FUNCTION_BLOCK FB_PUMP IMPLEMENTS I_PUMP
VAR //General
	{attribute 'instance-path'} 
  {attribute 'noinit'} 
	strInstancePath:									                      STRING;
	bInit: 												                          BOOL:=TRUE;
	strFullObjectPath: 								                      STRING;
	stEvent:											                          ST_EVENT;
	bAck:												                            BOOL;	
END_VAR
VAR   // From FB_init	
	itfLogEvents: 										                      I_HANDLE_EVENTS;
  itfOpMode:											                        I_OP_MODE; 
  itfOn:                                                  I_BINARY_OUTPUT;
END_VAR                                      				
VAR	// Step chain control                				
  eSeq, eLastSeq, eNextSeq:					                      E_SEQ_ENGINE; 
                  				
  //eActiveSeqState, eLastActiveSeqState:                 E_SEQ_GENERAL;
	(*
  iInternalSeqStateCase, iLastInternalSeqStateCase:       INT:=0;       
	tonDelay, tonTimeOut, tonStepTime:						          TON;
	tDelay:													                        TIME := T#100MS;
	tTimeOut:												                        TIME := T#100MS;
	tTimeOutExt:											                      TIME := T#100MS;
	bDelayActive, bTimeOutActiveQuit, bTimeOutActiveNoQuit:	BOOL;//Timer Option
	bActiveStep, bDebugAcitve, bDebugNext:					        BOOL;//Debug Option
	i:														                          INT;
 	iError:													                        INT; //ERROR-CODE                    	                   		
	listLastSteps:											                    ARRAY[0..49] OF ST_LAST_STEPS;	
	strExtraInfo:											                      STRING; 
	eStep_Type:												                      E_STEP_STATE_TYPE; 
	bDebugModeActive:										                    BOOL;   
	bWaitForBreakpoint:										                  BOOL;
	bBreakpointActive:										                  BOOL;
	bDebugResume:											                      BOOL;   
	listBreakpoint:											                    ARRAY[0..10] OF  INT;    
*)
i:														                            INT;
stSeqCtrlGeneral:											                    ST_SEQ_CTRL_GEN;     	
END_VAR                                             		
VAR                                                 		
	bMethodeFromExtStarted:									                BOOL;
	bMethodeFromExtActive:									                BOOL;
	bMethodeFromExtDone:									                  BOOL;
	strTemp:												                        STRING;
END_VAR   
VAR
  rLimit:                                                 REAL;
END_VAR                  	
VAR_TEMP                    	
	iTemp:										                              INT;
END_VAR

// Set FBs and Interfaces ready after switch internal step
IF stSeqCtrlGeneral.iInternalSeqStateCase <> stSeqCtrlGeneral.iLastInternalSeqStateCase AND NOT stSeqCtrlGeneral.bExitSetReadyState THEN
  IF TRUE
  //AND ...
  THEN
    stSeqCtrlGeneral.bExitSetReadyState := TRUE;
  ELSE
    RETURN;
  END_IF
END_IF

stSeqCtrlGeneral.strObject := F_CreateObjectName(strInstancePath);

// First method call
_m_SequenceManager();
//_m_SaveLastStep();

CASE eSeq OF 
  E_SEQ_VALVE.BASE:;
  
	E_SEQ_ENGINE.INIT: _m_Seq_INIT();
		IF TRUE
		AND (stSeqCtrlGeneral.eActiveSeqState = E_SEQ_GENERAL.DONE) 
		THEN
			eSeq := E_SEQ_ENGINE.BASE;
		END_IF
		
	E_SEQ_ENGINE.SETUP:;
  
	// Process
  E_SEQ_ENGINE.ON: _m_Seq_ON();
    IF TRUE
		AND (stSeqCtrlGeneral.eActiveSeqState = E_SEQ_GENERAL.DONE) 
		THEN
			eSeq := E_SEQ_VALVE.BASE;
		END_IF
    
  E_SEQ_ENGINE.OFF: _m_Seq_OFF();
    IF TRUE
		AND (stSeqCtrlGeneral.eActiveSeqState = E_SEQ_GENERAL.DONE) 
		THEN
			eSeq := E_SEQ_VALVE.BASE;
		END_IF

  // End
	E_SEQ_ENGINE.END:;
	E_SEQ_ENGINE.ERROR_SEQ:;	
END_CASE

strTemp:=TO_STRING(eSeq);

METHOD PRIVATE _m_DebugManager
VAR_INPUT
	iStepID: int;
END_VAR
IF TRUE
AND THIS^.stSeqCtrlGeneral.bDebugModeActive 
AND NOT THIS^.stSeqCtrlGeneral.bActiveStep
THEN


THIS^.stSeqCtrlGeneral.bBreakpointActive:=FALSE;

FOR i:=0 TO 10 DO
	
	IF TRUE
	AND iStepID=THIS^.stSeqCtrlGeneral.listBreakpoint[i] 
	AND iStepID<>0
	THEN
		EXIT;
	END_IF
END_FOR
IF (i<=10) THEN
	THIS^.stSeqCtrlGeneral.bBreakpointActive:=TRUE;
END_IF

END_IF
END_METHOD

METHOD PRIVATE _m_Delay : BOOL
VAR_INPUT
	DelayTime:	TIME;
END_VAR
THIS^.stSeqCtrlGeneral.bDelayActive:=TRUE;
THIS^.stSeqCtrlGeneral.tDelay:=DelayTime;
_m_Delay:=FALSE;
IF THIS^.stSeqCtrlGeneral.tonDelay.Q THEN
	_m_Delay:=TRUE;
END_IF
END_METHOD

METHOD PRIVATE _m_GeneralStepSetting : BOOL
VAR_INPUT
	StepType:			    	E_STEP_STATE_TYPE;
	InfoTextID:					STRING(20);
	EnableDebug:	   			BOOL;	
	
END_VAR
IF THIS^.stSeqCtrlGeneral.bActiveStep THEN
	THIS^.stSeqCtrlGeneral.eStep_Type:=StepType;
	THIS^.stSeqCtrlGeneral.strExtraInfo:= GenLib.F_RET_TXTLIST_ENTRY(strPortNr:='851',strID:='',strTxtLstName:=InfoTextID);
END_IF
END_METHOD

METHOD PRIVATE _m_SaveLastStep : BOOL
VAR_INPUT
END_VAR
VAR
	i: dint;
END_VAR
IF NOT THIS^.stSeqCtrlGeneral.bActiveStep THEN
	
	FOR i:=49 TO 1 BY -1 DO
			stSeqCtrlGeneral.listLastSteps[i].strStepName:=stSeqCtrlGeneral.listLastSteps[i-1].strStepName;
			stSeqCtrlGeneral.listLastSteps[i].tStepTime:=stSeqCtrlGeneral.listLastSteps[i-1].tStepTime;
			stSeqCtrlGeneral.listLastSteps[i].tDelayTime:=stSeqCtrlGeneral.listLastSteps[i-1].tDelayTime;
	END_FOR
	stSeqCtrlGeneral.listLastSteps[0].strStepName:=TO_STRING(THIS^.eSeq);
	stSeqCtrlGeneral.listLastSteps[1].tStepTime:=THIS^.stSeqCtrlGeneral.tonStepTime.ET;
	stSeqCtrlGeneral.listLastSteps[1].tStepTime:=THIS^.stSeqCtrlGeneral.tonDelay.ET;
ELSE
	stSeqCtrlGeneral.listLastSteps[0].tStepTime:=THIS^.stSeqCtrlGeneral.tonStepTime.ET;
	stSeqCtrlGeneral.listLastSteps[0].tDelayTime:=THIS^.stSeqCtrlGeneral.tonDelay.ET;	
END_IF
END_METHOD

METHOD PRIVATE _m_Seq_INIT : BOOL
VAR
  ActiveSeq: STRING;
END_VAR
//THIS^._m_GeneralStepSetting(StepType:=E_STEP_STATE_TYPE.INIT,
ActiveSeq := TO_STRING(THIS^.eSeq);

CASE THIS^.stSeqCtrlGeneral.eActiveSeqState OF
E_SEQ_GENERAL.READY:;

	
E_SEQ_GENERAL.EXECUTE:;
	IF TRUE
	THEN
		THIS^.stSeqCtrlGeneral.eActiveSeqState := E_SEQ_GENERAL.RESET;
	END_IF
  
E_SEQ_GENERAL.RESET:;
	stSeqCtrlGeneral.iInternalSeqStateCase := 0;
	IF TRUE
	THEN
		THIS^.stSeqCtrlGeneral.eActiveSeqState := E_SEQ_GENERAL.BUSY;
	END_IF
  
E_SEQ_GENERAL.BUSY:;
	CASE THIS^.stSeqCtrlGeneral.iInternalSeqStateCase OF
    0:  // Reset engine
      IF TRUE 
			THEN 
        THIS^.itfOn.M_Reset();
        THIS^.stSeqCtrlGeneral.iInternalSeqStateCase := 1000;
			END_IF
      
	ELSE
		THIS^.stSeqCtrlGeneral.eActiveSeqState := E_SEQ_GENERAL.DONE;  
	END_CASE
	THIS^.stSeqCtrlGeneral.strExtraInfo := CONCAT('Internal state: ', TO_STRING(THIS^.stSeqCtrlGeneral.iInternalSeqStateCase));

E_SEQ_GENERAL.DONE:;

E_SEQ_GENERAL.ERROR:;

E_SEQ_GENERAL.TIME_OUT:; 
IF TRUE
AND THIS^.stSeqCtrlGeneral.bTimeOutActiveQuit 
THEN
  THIS^.stSeqCtrlGeneral.strExtraInfo := 'Bitte quittieren und erneut testen';
  IF TRUE
  //AND itfOpMode.P_QUIT
  THEN
    THIS^.stSeqCtrlGeneral.eActiveSeqState := E_SEQ_GENERAL.EXECUTE;
	END_IF
  
END_IF

ELSE
  THIS^.stSeqCtrlGeneral.eActiveSeqState := E_SEQ_GENERAL.ERROR;
END_CASE
END_METHOD

METHOD _m_Seq_OFF : BOOL
VAR
  ActiveSeq: STRING;
END_VAR
//THIS^._m_GeneralStepSetting(StepType:=E_STEP_STATE_TYPE.INIT,
ActiveSeq := TO_STRING(THIS^.eSeq);

CASE THIS^.stSeqCtrlGeneral.eActiveSeqState OF
E_SEQ_GENERAL.READY:;

	
E_SEQ_GENERAL.EXECUTE:;
	IF TRUE
	THEN
		THIS^.stSeqCtrlGeneral.eActiveSeqState := E_SEQ_GENERAL.RESET;
	END_IF
  
E_SEQ_GENERAL.RESET:;
	stSeqCtrlGeneral.iInternalSeqStateCase := 0;
	IF TRUE
	THEN
		THIS^.stSeqCtrlGeneral.eActiveSeqState := E_SEQ_GENERAL.BUSY;
	END_IF
  
E_SEQ_GENERAL.BUSY:;
	CASE THIS^.stSeqCtrlGeneral.iInternalSeqStateCase OF
    0:  // Engine off
      IF TRUE 
			THEN 
        THIS^.itfOn.M_Reset();
        THIS^.stSeqCtrlGeneral.iInternalSeqStateCase := 1000;
			END_IF
      
	ELSE
		THIS^.stSeqCtrlGeneral.eActiveSeqState := E_SEQ_GENERAL.DONE;  
	END_CASE
	THIS^.stSeqCtrlGeneral.strExtraInfo := CONCAT('Internal state: ', TO_STRING(THIS^.stSeqCtrlGeneral.iInternalSeqStateCase));

E_SEQ_GENERAL.DONE:;

E_SEQ_GENERAL.ERROR:;

E_SEQ_GENERAL.TIME_OUT:; 
IF TRUE
AND THIS^.stSeqCtrlGeneral.bTimeOutActiveQuit 
THEN
  THIS^.stSeqCtrlGeneral.strExtraInfo := 'Bitte quittieren und erneut testen';
  IF TRUE
  //AND itfOpMode.P_QUIT
  THEN
    THIS^.stSeqCtrlGeneral.eActiveSeqState := E_SEQ_GENERAL.EXECUTE;
	END_IF
  
END_IF

ELSE
  THIS^.stSeqCtrlGeneral.eActiveSeqState := E_SEQ_GENERAL.ERROR;
END_CASE
END_METHOD

METHOD PRIVATE _m_Seq_ON : BOOL
VAR
  ActiveSeq: STRING;
END_VAR
//THIS^._m_GeneralStepSetting(StepType:=E_STEP_STATE_TYPE.INIT,
ActiveSeq := TO_STRING(THIS^.eSeq);

CASE THIS^.stSeqCtrlGeneral.eActiveSeqState OF
E_SEQ_GENERAL.READY:;

	
E_SEQ_GENERAL.EXECUTE:;
	IF TRUE
	THEN
		THIS^.stSeqCtrlGeneral.eActiveSeqState := E_SEQ_GENERAL.RESET;
	END_IF
  
E_SEQ_GENERAL.RESET:;
	stSeqCtrlGeneral.iInternalSeqStateCase := 0;
	IF TRUE
	THEN
		THIS^.stSeqCtrlGeneral.eActiveSeqState := E_SEQ_GENERAL.BUSY;
	END_IF
  
E_SEQ_GENERAL.BUSY:;
	CASE THIS^.stSeqCtrlGeneral.iInternalSeqStateCase OF
    0:  // Engine on
      IF TRUE 
			THEN 
        THIS^.itfOn.M_Set();
        THIS^.stSeqCtrlGeneral.iInternalSeqStateCase := 1000;
			END_IF
      
	ELSE
		THIS^.stSeqCtrlGeneral.eActiveSeqState := E_SEQ_GENERAL.DONE;  
	END_CASE
	THIS^.stSeqCtrlGeneral.strExtraInfo := CONCAT('Internal state: ', TO_STRING(THIS^.stSeqCtrlGeneral.iInternalSeqStateCase));

E_SEQ_GENERAL.DONE:;

E_SEQ_GENERAL.ERROR:;

E_SEQ_GENERAL.TIME_OUT:; 
IF TRUE
AND THIS^.stSeqCtrlGeneral.bTimeOutActiveQuit 
THEN
  THIS^.stSeqCtrlGeneral.strExtraInfo := 'Bitte quittieren und erneut testen';
  IF TRUE
  //AND itfOpMode.P_QUIT
  THEN
    THIS^.stSeqCtrlGeneral.eActiveSeqState := E_SEQ_GENERAL.EXECUTE;
	END_IF
  
END_IF

ELSE
  THIS^.stSeqCtrlGeneral.eActiveSeqState := E_SEQ_GENERAL.ERROR;
END_CASE
END_METHOD

METHOD PRIVATE _m_SequenceManager
VAR_INPUT
END_VAR
IF FALSE
//AND THIS^.eActiveSeqState=DONE 
AND eLastSeq<>eSeq
THEN
	IF THIS^.stSeqCtrlGeneral.eActiveSeqState<>E_SEQ_GENERAL.EXECUTE THEN
		THIS^.stSeqCtrlGeneral.eActiveSeqState:=E_SEQ_GENERAL.READY;
	END_IF
END_IF

eSeq := eNextSeq;

//DelayTimer und TimeOut Timer verwalten
stSeqCtrlGeneral.bActiveStep:=	TRUE
				AND eLastSeq					=	eSeq
				AND stSeqCtrlGeneral.eLastActiveSeqState			=	stSeqCtrlGeneral.eActiveSeqState
				AND	stSeqCtrlGeneral.iLastInternalSeqStateCase	=	stSeqCtrlGeneral.iInternalSeqStateCase
				;
			
IF NOT stSeqCtrlGeneral.bActiveStep THEN
	stSeqCtrlGeneral.bDelayActive:=FALSE;
	stSeqCtrlGeneral.bTimeOutActiveQuit:=FALSE;
	stSeqCtrlGeneral.bTimeOutActiveNoQuit:=FALSE;
  THIS^.stSeqCtrlGeneral.strExtraInfo:='';
END_IF

_m_SaveLastStep();
stSeqCtrlGeneral.tonDelay	(IN:=stSeqCtrlGeneral.bActiveStep AND stSeqCtrlGeneral.bDelayActive, 		PT:=stSeqCtrlGeneral.tDelay);
stSeqCtrlGeneral.tonTimeOut	(IN:=stSeqCtrlGeneral.bActiveStep AND (stSeqCtrlGeneral.bTimeOutActiveNoQuit OR stSeqCtrlGeneral.bTimeOutActiveQuit), 	PT:=stSeqCtrlGeneral.tTimeOut);
stSeqCtrlGeneral.tonStepTime	(IN:= stSeqCtrlGeneral.bActiveStep, PT:= T#24H);

IF stSeqCtrlGeneral.tonTimeOut.Q  THEN
	stSeqCtrlGeneral.eActiveSeqState:=E_SEQ_GENERAL.TIME_OUT;
END_IF

IF stSeqCtrlGeneral.iError<>0 THEN
	eSeq:=E_SEQ_ENGINE.ERROR_SEQ;
END_IF



eLastSeq					:=	eSeq;
stSeqCtrlGeneral.eLastActiveSeqState			:=	stSeqCtrlGeneral.eActiveSeqState;
stSeqCtrlGeneral.iLastInternalSeqStateCase	:=	stSeqCtrlGeneral.iInternalSeqStateCase;

// Reset set ready state
IF THIS^.stSeqCtrlGeneral.bExitSetReadyState THEN
  THIS^.stSeqCtrlGeneral.bExitSetReadyState := FALSE;
END_IF
END_METHOD

METHOD PRIVATE _m_TimeOut : BOOL
VAR_INPUT
	bTimeoutActiveToQuit:	BOOL;
	bTimeOutActiveNoQuit:	BOOL;
	tTimeOut:				TIME;	
END_VAR
THIS^.stSeqCtrlGeneral.bTimeOutActiveQuit:=	bTimeoutActiveToQuit;
THIS^.stSeqCtrlGeneral.bTimeOutActiveNoQuit:=	bTimeOutActiveNoQuit;
THIS^.stSeqCtrlGeneral.tTimeOut:=			tTimeOut;
_m_TimeOut:=FALSE;
IF THIS^.stSeqCtrlGeneral.tonTimeOut.Q THEN
	_m_TimeOut:=TRUE;
END_IF
END_METHOD

METHOD FB_init : BOOL
VAR_INPUT
	bInitRetains : BOOL; // if TRUE, the retain variables are initialized (warm start / cold start)
	bInCopyCode : BOOL;  // if TRUE, the instance afterwards gets moved into the copy code (online change)
  
  itfLogEvents: 										                      I_HANDLE_EVENTS;
  itfOpMode:											                        I_OP_MODE; 
  itfOn:                                                  I_BINARY_OUTPUT;
END_VAR
THIS^.itfLogEvents := itfLogEvents;
THIS^.itfOpMode := itfOpMode;
THIS^.itfOn := itfOn;
END_METHOD

METHOD M_Off : BOOL
M_Off := THIS^.stSeqCtrlGeneral.eActiveSeqState = E_SEQ_GENERAL.DONE;

// Assign input

// General
IF THIS^.stSeqCtrlGeneral.eActiveSeqState = E_SEQ_GENERAL.READY THEN
  THIS^.eNextSeq := E_SEQ_ENGINE.OFF;
  THIS^.stSeqCtrlGeneral.eActiveSeqState := E_SEQ_GENERAL.EXECUTE;
END_IF
END_METHOD

METHOD M_On : BOOL
M_On := THIS^.stSeqCtrlGeneral.eActiveSeqState = E_SEQ_GENERAL.DONE;

// Assign input

// General
IF THIS^.stSeqCtrlGeneral.eActiveSeqState = E_SEQ_GENERAL.READY THEN
  THIS^.eNextSeq := E_SEQ_ENGINE.ON;
  THIS^.stSeqCtrlGeneral.eActiveSeqState := E_SEQ_GENERAL.EXECUTE;
END_IF
END_METHOD

METHOD M_Reset : BOOL
VAR_INPUT
END_VAR
M_Reset := THIS^.stSeqCtrlGeneral.eActiveSeqState = E_SEQ_GENERAL.DONE;

// Assign input

// General
IF THIS^.stSeqCtrlGeneral.eActiveSeqState = E_SEQ_GENERAL.READY THEN
  THIS^.eNextSeq := E_SEQ_ENGINE.INIT;
  THIS^.stSeqCtrlGeneral.eActiveSeqState := E_SEQ_GENERAL.EXECUTE;
END_IF
END_METHOD

{warning 'Methodenimplementierung hinzufügen'}
(*=== Method: M_Run  ============================================

 @brief: Here is the global code (Timer, Event, Flange,...)*)
METHOD M_Run
END_METHOD

METHOD M_SetReady : BOOL
VAR_INPUT
END_VAR
M_SetReady := stSeqCtrlGeneral.eActiveSeqState = E_SEQ_GENERAL.READY;

THIS^.stSeqCtrlGeneral.eActiveSeqState := E_SEQ_GENERAL.READY;
END_METHOD

{warning 'Eigenschaftenimplementierung hinzufügen'}
PROPERTY P_Busy : BOOL
GET
IF stSeqCtrlGeneral.eActiveSeqState = E_SEQ_GENERAL.READY THEN
  P_Busy := FALSE;
ELSE
  P_Busy := TRUE;
END_IF
END_GET
END_PROPERTY

{warning 'Eigenschaftenimplementierung hinzufügen'}
(*=== Property: P_Event  ============================================

 @param [set]: 	Set the Structure "ST_EVENT" from another Object
 @param [get]: 	Return the Structure "ST_EVENT", it contains the actual 
					event of the Object *)
PROPERTY P_Event : GenLib.ST_EVENT
GET
END_GET
SET
END_SET
END_PROPERTY

{warning 'Eigenschaftenimplementierung hinzufügen'}
(*=== Property: P_FullObjectPath  ============================================

 @param [set]: 	Set the Object Path (Clear String of Object)
 @param [get]: 	Return the Objectpath *)
PROPERTY P_FullObjectPath : STRING
GET
END_GET
SET
END_SET
END_PROPERTY

{warning 'Eigenschaftenimplementierung hinzufügen'}
(*=== Property: P_Global_Ack  ============================================

 @param [set]: 	Set the Bit for Ack from another Object
 @param [get]: 	Return the state of Ack Bit*)
PROPERTY P_Global_Ack : BOOL
GET
END_GET
SET
END_SET
END_PROPERTY

{warning 'Eigenschaftenimplementierung hinzufügen'}
(*=== Property: P_GlobalID  ============================================

 @param [set]: 	-
 @param [get]: 	Return the string of instance path*)
PROPERTY P_GlobalID : STRING
GET
END_GET
END_PROPERTY

{warning 'Eigenschaftenimplementierung hinzufügen'}
PROPERTY P_ReadyState : BOOL
GET
P_ReadyState := THIS^.stSeqCtrlGeneral.eActiveSeqState = E_SEQ_GENERAL.READY;
END_GET
END_PROPERTY

//{​​​​attribute 'monitoring' := 'call'}​​​​
PROPERTY P_State : BOOL
GET
P_State := THIS^.itfOn.P_State;
END_GET
END_PROPERTY

END_FUNCTION_BLOCK

(* stored: Version 1.1.0.1, ProductVersion 3.1.4024.12
   POU FB_PUMP: Id {1fad881b-aced-41bf-a3e0-db3cfecbbe0b}, SpecialFunc None
   Folder PRIVAT: Id {cfb1d420-05c5-4380-9897-4b71c118e2ed}
   Folder SEQUENCE: Id {5c37ff53-acd0-4e21-b829-2333928dc10e}
   Method _m_DebugManager: Id {92125b30-04be-4215-bb5f-61c785e04565}
   Method _m_Delay: Id {3d6d0246-9a0a-4935-b7e9-20778df12c39}
   Method _m_GeneralStepSetting: Id {4ae89094-31d7-4a9b-9c2b-4f3b99719ef2}
   Method _m_SaveLastStep: Id {a754827d-dfc7-47e1-8eca-8d5f579d9234}
   Method _m_Seq_INIT: Id {9279831e-4bc8-4605-a763-3c88a6722dd2}
   Method _m_Seq_OFF: Id {ef7435cb-9f84-4219-a4f5-8d8f516e0375}
   Method _m_Seq_ON: Id {87be2655-a393-4e92-bc97-8d91dec91b96}
   Method _m_SequenceManager: Id {4ae31ade-5d80-48eb-8ecd-3104089b15dd}
   Method _m_TimeOut: Id {1dd43463-79e2-4de3-95be-3c8a8cbeaed6}
   Method FB_init: Id {64a216f9-629f-45cd-a0bc-8c0590c76c60}
   Method M_Off: Id {ccd28b34-8f1d-439a-9787-717b494f4166}
   Method M_On: Id {b528b287-cab7-494e-b7b9-79a6ef41bb31}
   Method M_Reset: Id {38836e02-00c9-4569-b784-9a060dad2092}
   Method M_Run: Id {469cad35-8e10-49b1-8383-05e0018e402f}
   Method M_SetReady: Id {f04bb520-cfbc-420c-9812-686a276504b2}
   Property P_Busy: Id {8b196493-34a1-4fd3-a11c-652c3fdc5b66}
   Get Get: Id {498e56d9-e5b5-4e10-935c-b97e9e850b2d}
   Property P_Event: Id {3eefe73a-c192-4e95-98f3-63e2030911ae}
   Get Get: Id {777c99b3-8e91-488c-b25a-a90765f4cbbf}
   Set Set: Id {78928900-1ce4-4b5e-a173-48be0cf217e0}
   Property P_FullObjectPath: Id {6a32912f-208b-4b3f-bcf1-7f3ba708733c}
   Get Get: Id {f00e55a8-601a-4ada-82a9-84c0e8584e73}
   Set Set: Id {ec559945-7aca-44ef-b28f-7367395851a7}
   Property P_Global_Ack: Id {18caf017-56bb-4efc-9d34-7e5b37fa8044}
   Get Get: Id {2225e31f-7556-4b9f-85f7-9ffdf1cf0387}
   Set Set: Id {3b7abd5d-b135-4990-90b1-bd16451896d7}
   Property P_GlobalID: Id {151c8eb4-819c-4ffe-9847-e4ce80d9465d}
   Get Get: Id {065f57f2-38b9-4488-b26a-b462dac41df5}
   Property P_ReadyState: Id {47250e69-3aba-47f5-94e1-d1922b0e4916}
   Get Get: Id {8256e3f4-0849-49e0-8333-73da6a373c13}
   Property P_State: Id {6e2ede0c-1aaf-447c-8d78-4f92f315d457}
   Get Get: Id {d1289add-17f6-4fdc-87bb-d7aedaef0c61} *)
